/// Function convert EtherCat master device state into an text
FUNCTION F_Diagnostic_EcMasterDeviceState : WSTRING(80)
VAR_INPUT
	/// Function input
	nDeviceState			:UINT;
END_VAR
VAR
END_VAR

CASE nDeviceState OF
	// Link error
	16#1:
		F_Diagnostic_EcMasterDeviceState := "EtherCat: Link error";
		
	// I/O locked after link error (I/O reset required)
	16#2:
		F_Diagnostic_EcMasterDeviceState := "EtherCat: I/O locked after link error (I/O reset required)";
		
	// Link error (redundancy adapter)
	16#4:
		F_Diagnostic_EcMasterDeviceState := "EtherCat: Link error (redundancy adapter)";
		
	// Missing one frame (redundancy mode)
	16#8:
		F_Diagnostic_EcMasterDeviceState := "EtherCat: Missing one frame (redundancy mode)";
		
	// Out of send resources (I/O reset required)
	16#10:
		F_Diagnostic_EcMasterDeviceState := "EtherCat: Out of send resources (I/O reset required)";
		
	// Watchdog triggered
	16#20:
		F_Diagnostic_EcMasterDeviceState := "EtherCat: Watchdog triggered";
		
	// Ethernet driver (miniport) not found
	16#40:
		F_Diagnostic_EcMasterDeviceState := "EtherCat: Ethernet driver (miniport) not found";
		
	// I/O reset active
	16#80:
		F_Diagnostic_EcMasterDeviceState := "EtherCat: I/O reset active";
		
	// At least one device in "INIT" state
	16#100:
		F_Diagnostic_EcMasterDeviceState := "EtherCat: At least one device in INIT state";
		
	// At least one device in "PRE-OP" state
	16#200:
		F_Diagnostic_EcMasterDeviceState := "EtherCat: At least one device in PRE-OP state";
		
	// At least one device in "SAFE-OP" state
	16#400:
		F_Diagnostic_EcMasterDeviceState := "EtherCat: At least one device in SAFE-OP state";
		
	// At least one device indicates an error state
	16#800:
		F_Diagnostic_EcMasterDeviceState := "EtherCat: At least one device indicates an error state";
		
	// DC not in sync
	16#1000:
		F_Diagnostic_EcMasterDeviceState := "EtherCat: DC not in sync";
		
	ELSE 
		F_Diagnostic_EcMasterDeviceState := WCONCAT("EtherCat error: ", UINT_TO_WSTRING(nDeviceState));
END_CASE

END_FUNCTION

(* stored: Version 1.1.0.1, ProductVersion 3.1.4024.11
   POU F_Diagnostic_EcMasterDeviceState: Id {e3672b09-bc1c-4880-a6a7-d28936e7dc50}, SpecialFunc None *)
